FUNCTION_BLOCK FB_Spindle
VAR_INPUT
	Enable	: BOOL; // Enable the servo
	SetVelo	: REAL;	// Speed in RPMs
END_VAR
VAR_IN_OUT
	data	: ST_Spindle;	// Ethernet IP data
END_VAR
VAR_OUTPUT
	ActVelo	: REAL;	//Speed in RPMs
	Ready	: BOOL; // Servo ready to move
	Error	: UINT; // 0 = OK, 1 = not connected
END_VAR
VAR
	rTargetVel	: REAL;	
	fbTrigEnable	: BOOL;	
	iState	: DINT;	
	fbDelay	: TON;
	bRunDelay	: BOOL;
END_VAR

IF NOT Enable THEN
	iState := 0;
END_IF
// Scale target rpm
rTargetVel := SCALE_R(
				X:= SetVelo, 
				I_LO:= -15000, 
				I_HI:= 15000, 
				O_LO:= -30000, 
				O_HI:= 30000);
				
fbDelay(IN:= bRunDelay, PT:= T#1000MS, Q=> , ET=> );				

CASE iState OF
0:	// Default, set all output to 0
	MEMSET(ADR(data.out.flags), 0, SIZEOF(data.out.flags));
	bRunDelay := FALSE;
	IF Enable THEN
		iState := 10;
	END_IF
10:
	IF data.in.flags.DriveError THEN
		data.out.flags.ResetFault := TRUE;
		iState := 20;	// Reset state
	ELSE			
		iState := 100;	// OK to run
	END_IF	
20:
	data.out.flags.ServoEnable := FALSE;
	data.out.flags.ResetFault := data.in.flags.DriveError;
	bRunDelay := TRUE;	// Don't try to power on for at least a second
	IF NOT data.in.flags.DriveError AND fbDelay.Q THEN
		iState := 100;
		bRunDelay := FALSE;
	END_IF
	
100:
	data.out.flags.ServoEnable := TRUE;
	data.out.SpindleSpeed := TO_INT(rTargetVel);
	
	IF data.in.flags.DriveError THEN
		iState := 999;
	END_IF
	
999: // Stay in fault state until error can be examined
	data.out.flags.ServoEnable := FALSE;
	;
END_CASE


Error := TO_UINT(data.in.flags.DriveError);
Ready := Error = 0 AND data.in.flags.Contactor1 AND data.in.flags.Contactor2 AND data.DevState = 0;


IF data.in.flags.RpmLT5 THEN
	ActVelo := 0;
ELSE
	ActVelo := SCALE_R(
		X:= data.in.SpindleSpeed, 
		I_LO:= -30000, 
		I_HI:= 30000, 
		O_LO:= -15000, 
		O_HI:= 15000);
END_IF

METHOD OpcuaMonitor : BOOL
VAR_INPUT
END_VAR
VAR_IN_OUT
	Data	: ST_SpindleControl;
END_VAR
VAR_OUTPUT
	Error	: BOOL;
END_VAR
VAR_INST
	fbHbMonitor	: FB_HeartbeatMonitor;
END_VAR
fbHbMonitor(CLK:= Data.status.input.Heartbeat, PT:= T#2.5S, Q=> );

IF NOT fbHbMonitor.Q THEN
	MEMSET(ADR(Data.input), 0, SIZEOF(Data.input));
	Error := TRUE;
ELSE
	Error := FALSE;
END_IF
END_METHOD

END_FUNCTION_BLOCK

(* stored: Version 1.1.0.1, ProductVersion 3.1.4024.9
   POU FB_Spindle: Id {eefa1b23-964a-4427-b06c-af0370dca8a6}, SpecialFunc None
   Method OpcuaMonitor: Id {563c18c7-eb09-469e-b42e-c17efa116a0d} *)
